(* CODESYS project FileOperation.project

Project tree, tasks and I/O mapping:
  Device : CODESYS Control for Raspberry Pi MC SL, CODESYS GmbH, order no. 2302000009, version 4.11.0.0
    application Application
      libraries: Standard, 3.5.18.0 (System); VisuDialogs, 4.5.0.0 (System); Visu Utils, 4.5.0.0 (System); CAA File, * (CAA Technical Workgroup)
      task MainTask (cyclic, interval t#20ms, priority 1, watchdog t#100ms x 1) calls TEST_FileFB, SK_FileDialogExec, Test_SK_FileDialogExec
      task VISU_TASK (cyclic, interval 100 ms, priority 31) calls VisuElems.Visu_Prg
      DialogTest/
        visualisation VS_TEST_SK_FileDialogExec
        program Test_SK_FileDialogExec [ST]
      Define/
        data type CharToStringBuffer
        data type CharCode
        data type AxisData
        data type TestCheck
        data type TestState
        data type FIX_TBL
        data type SK_FileSelectDialogVar
        data type SK_FileInfo
      FunctionBlockTest/
        program TEST_FileFB [ST]
      LIBs/
        function block SKFB_ReadFile [ST]
        function block SKFB_ReadFixTbl [ST]
        function block SKFB_WriteFile [ST]
        function block SKFB_WriteFixTbl [ST]
        program SK_FileDialogExec [ST]
        visualisation SKVS_FileSelectDialog
        function block SKFB_ListFilesInDir [ST]
    GPIOs_A_B : GPIOs A/B, 3S - Smart Software Solutions GmbH, version 4.11.0.0
        unmapped channels: digital inputs (GPIO0..GPIO31), digital outputs (GPIO0..GPIO31)
    Onewire
    Camera device
      <空>
    SPI
    I²C
    SoftMotion General Axis Pool
  text list GlobalTextList
*)

// Device/Application/Define/CharToStringBuffer
TYPE CharToStringBuffer :
UNION
	ValueBuffer: ARRAY [0..31] OF BYTE;
	ValueString: STRING;
END_UNION
END_TYPE

// Device/Application/Define/CharCode
{attribute 'qualified_only'}
{attribute 'strict'}
TYPE CharCode :
(
	NULL := 0,
	CR:= 16#0D,
	LF:= 16#0A,
	COMMA:= 16#2C	
);
END_TYPE

// Device/Application/Define/AxisData
TYPE AxisData :
STRUCT
	Value: ARRAY [0..5] OF REAL; 	//VX,VY,VZ,VA,VB,VC:REAL;
END_STRUCT
END_TYPE

// Device/Application/Define/TestCheck
TYPE TestCheck :

STRUCT
	State:TestState:= TestState.Wait;
	Msg:STRING;
END_STRUCT

END_TYPE

// Device/Application/Define/TestState
{attribute 'qualified_only'}
{attribute 'strict'}
TYPE TestState :
(
	Wait:=0, Exec:=1, Success:=10, Error:=-1
);
END_TYPE

// Device/Application/Define/FIX_TBL
TYPE FIX_TBL :
STRUCT
	Value:ARRAY[0..5,1..20] OF LREAL;
END_STRUCT
END_TYPE

// Device/Application/Define/SK_FileSelectDialogVar
TYPE SK_FileSelectDialogVar :
(*
	2024/08/02 SKVS_FileSelectDialogとやり取りする変数	
*)

STRUCT
	ListPath:STRING;//一覧で表示するパスの場所

	//FileData:ARRAY[1..SK_FileDialogExec.MAX_FILE_LISTING] OF SK_FileInfo;
	//FileCount:INT;
	Selected:INT;
	
	//Ok時に決定されたパス＋ファイル名
	//ResultPathFileName:STRING;
	////Ok時に決定されたファイル名(パスはない)
	ResultFileName:STRING;
	
	//Option_SaveMode:BOOL:=FALSE;  // 

	//Userが自由に設定できるフラグ
	//UserFlag:INT:=0;
	
	//----------------- 結果の取得 ----------------------
	
	//OKボタンで終了したらTRUE
	//DialogOK:BOOL;	
	
	//Cancelボタンで終了したらTRUE
	//DialogCancel:BOOL;
	
END_STRUCT

END_TYPE

// Device/Application/Define/SK_FileInfo
TYPE SK_FileInfo :
STRUCT
	FileName:STRING;
	FileSize:STRING;
	LastModifyDT:STRING;
END_STRUCT
END_TYPE

// Device/Application/FunctionBlockTest/TEST_FileFB
PROGRAM TEST_FileFB
(* ファイル関連のFBをテストするプログラム　*)

(* 
準備事項 RPi版 
Device-ファイルで、
ランタイム（右側）で、PlcLogicが カレントになるので、
/PlcLogic
  + /CNC_DATA
    + /LOG
    + /CONFIG
    + /GCODE

のフォルダを作製する。　
プログラムからは、　CNC_DATA/CONFIG/aaa.csv のようにアクセスする

*)

(* 
準備事項 HX版 
Device-ファイルで、
ランタイム（右側）で、SDCardが /に相当するので、
/SDCard
  + /CNC_DATA
    + /LOG
    + /CONFIG
    + /GCODE

のフォルダを作製する。
プログラムからは、　/media/sd-mmcblk0p1/CNC_DATA/CONFIG/aaa.csv のようにアクセスする
*)

VAR CONSTANT
	VAR_TBL_COUNT:INT:=20;	
	FilePath:STRING:= 'CNC_DATA/CONFIG/';	//RPi
	//FilePath:STRING:= '/media/sd-mmcblk0p1/CNC_DATA/CONFIG/';	//HITACHI HX
END_VAR	
	

VAR 	
	//GCode Table
	TBL_W:ARRAY [0..5(*AXIS*),1..VAR_TBL_COUNT] OF LREAL;
	TBL_R:ARRAY [0..5(*AXIS*),1..VAR_TBL_COUNT] OF LREAL;


	FBRead:SKFB_ReadFixTbl;
	CheckReadData:TestCheck;

	FBWriteLine:SKFB_WriteFile;
	WriteLineArray: ARRAY[0..1] OF STRING;
	CheckWriteLine:TestCheck;

	FBWrite:SKFB_WriteFixTbl;
	CheckWriteData:TestCheck;
	
	i_row,i_axis:INT;
	//Initialized:BOOL:=FALSE;
	
END_VAR


// テストシーケンス


IF (CheckWriteLine.State=TestState.Wait) THEN
	CheckWriteLine.State:= TestState.Exec;
END_IF

IF (CheckWriteLine.State=TestState.Success) AND (CheckWriteData.State= TestState.Wait) THEN
	CheckWriteData.State:=TestState.Exec;
END_IF

IF (CheckWriteData.State=TestState.Success) AND (CheckReadData.State= TestState.Wait)THEN
	CheckReadData.State:=TestState.Exec;
END_IF

(*
IF (CheckReadData.State= TestState.Wait)THEN
	CheckReadData.State:=TestState.Exec;
END_IF
*)

//--------------------   Exec Function Block   --------------------------


IF (CheckReadData.State= TestState.Exec) THEN 
	FBRead(
		pData:=ADR(TBL_R),
		DataCount:=20,
		FileName:='TEST.CSV',
		Path:=FilePath,
		xExec:=TRUE
	);
	IF(FBRead.xDone) THEN
		FBRead(xExec:=FALSE);
		CheckReadData.Msg:= FBRead.Msg;
		CheckReadData.State := TestState.Success;	
	END_IF
	IF (FBRead.xError) THEN
		FBRead(xExec:=FALSE);	
		CheckReadData.Msg:= FBRead.Msg;
		CheckReadData.State := TestState.Error;	
	END_IF
	
END_IF

IF (CheckWriteData.State= TestState.Exec) THEN
	// SetTestData
	FOR i_row:=1 TO VAR_TBL_COUNT DO
		FOR i_axis:=0 TO 5 DO
			TBL_W[i_axis,i_row]:= i_row*10+ i_axis;
		END_FOR
	END_FOR
	
	FBWrite(
		pData:=ADR(TBL_W),
		//DataCount:=20,
		FileName:='TEST.CSV',
		Path:=FilePath,
		xExec:=TRUE
	);
	IF(FBWrite.xDone) THEN
		FBWrite(xExec:=FALSE);
		CheckWriteData.Msg:= CheckWriteData.Msg;
		CheckWriteData.State := TestState.Success;	
	END_IF
	IF (FBWrite.xError) THEN
		FBWrite(xExec:=FALSE);	
		CheckWriteData.Msg:= CheckWriteData.Msg;
		CheckWriteData.State := TestState.Error;	
	END_IF
	
END_IF


IF CheckWriteLine.State= TestState.Exec THEN
	WriteLineArray[0]:='123456789$0D$0A';
	WriteLineArray[1]:='ABCDEFG$0D$0A';

	FbWriteLine(
		pWriteLines:= ADR(WriteLineArray),
		WriteLinesCount:=2,
		FilePathName:=CONCAT(FilePath,'1.TXT'),
		xExec:=TRUE
	);
	
	IF FbWriteLine.xDone THEN
		CheckWriteLine.Msg:= FbWriteLine.Msg;
		CheckWriteLine.State := TestState.Success;	
		FbWriteLine(xExec:=FALSE);
	END_IF
	IF FbWriteLine.xError THEN
		CheckWriteLine.Msg:= FbWriteLine.Msg;
		CheckWriteLine.State := TestState.Error;	
		FbWriteLine(xExec:=FALSE);
	END_IF
		
END_IF

END_PROGRAM

// Device/Application/LIBs/SKFB_ReadFixTbl
FUNCTION_BLOCK SKFB_ReadFixTbl
(*
	2024/08/02
	FixテーブルのCSVファイルを指定のバッファに読み込む
	注意:CAA File 3.5.15 を使っているため、PCエミュレーターには対応していない。　実機に転送して実行すること	
	ファイルバッファREAD_FILE_BUFFERを確保して読み込むのでファイルの大きさに注意(改善点)
*)

// Interface Variables ---------------------------------------------------

VAR_INPUT
	FileName:STRING:='';	//パスは含まない	
	Path:STRING := '';
	pData:POINTER TO FIX_TBL:=0; //データメモリへのポインタ
	DataCount:UINT:=0;  // ファイルにデータメモリ以上のデータがある場合は無視されます

	xExec:BOOL:=FALSE;	//実行・維持フラグ	
	PARSE_CHAR_COUNT:UINT:= 256;   //一度のサイクル処理でパースする文字数

END_VAR

VAR_OUTPUT
	xDone:BOOL;
	xError:BOOL;
	Msg:STRING;

	ReadRowCount: DINT; 		//読み込んだデータ数
	ExecState: INT:= stInit;	//現在の実行状況
	//DataHeader: STRING;	
END_VAR


VAR CONSTANT
	//State
	stInit:INT:=0;
	stWait:INT := 1; 
	stFileToBuffer:INT:=2;

	stParseHeader:INT:=3;
	stParseData:INT:=4;

	//Result
	stDone:INT := 100;
	stError:INT:= 999;

	//ファイルバッファ
	READ_FILE_BUFFER:UINT:=1024*16;  //バッファ	16K

END_VAR

// Implementation Variables ---------------------------------------------------


VAR
	
	FbFileRead:SKFB_ReadFile;
	RawBuff: ARRAY [0..READ_FILE_BUFFER-1] OF BYTE;	
	i_RawBuff,i_add:UINT;
	CurrBuff:BYTE;
	
	i_TempChar, i_Row, i_Axis, i_TempCharClear: INT;

	TmpCharBuffer: CharToStringBuffer;
END_VAR

CASE ExecState OF
	
	stInit:
		//初期化
		xDone:=FALSE;
		xError:=FALSE;
		Msg:='';
		FbFileRead(xExec := FALSE);
		ExecState:= stWait;
		ReadRowCount:=-1;
		
	stWait:
		IF xExec THEN
			//Exec状態になった　-->Check Input Variables 
			IF pData=0 THEN
				Msg:='pData is not set.';
				ExecState:=stError;
			ELSIF DataCount=0 THEN
				Msg:='ReadBufferSize is not set.';
				ExecState:=stError;
			ELSIF Path='' THEN
				Msg:='Path is not set.';
				ExecState:=stError;
			ELSIF FileName='' THEN
				Msg:='Path is not set.';
				ExecState:=stError;
			ELSE
				//Proceed Next State
				ExecState:= stFileToBuffer;
			END_IF
		END_IF
	
	stFileToBuffer:	// File Open
		
		FbFileRead(
			xExec:= TRUE, 
			pReadBuffer:= 		ADR(RawBuff),
			ReadBufferSize:= 	READ_FILE_BUFFER,
			FilePathName:= CONCAT(Path,FileName)
		);
	
		// Until Done or Error
		IF FbFileRead.xDone THEN
			FbFileRead(xExec := FALSE);
	
			//出力メモリのクリア
			FOR i_Row:=1 TO 20 DO
				FOR i_Axis:=0 TO 5 DO 
					pData^.Value[i_Axis,i_Row]:=0;			
				END_FOR
			END_FOR
			
			ExecState := stParseHeader;
			i_RawBuff := 0;
			i_TempChar := 0;
			i_Row := 1;
			i_Axis := 0;
			//DataHeader:='';
			
			//Clear Buffer
			FOR i_TempCharClear := 0 TO 31 DO
				TmpCharBuffer.ValueBuffer[i_TempCharClear] := 0;
			END_FOR
	
		ELSIF FbFileRead.xError THEN
			Msg:= CONCAT('FileToBuffer:',FbFileRead.Msg);
			FbFileRead(xExec := FALSE);
	
			ExecState := stError;
		END_IF

	StParseHeader:	// Skip DataTitle
		ExecState:=stParseData;

(*
	//PARSE_CHAR_COUNTづつ処理
	FOR i_add:=0 TO PARSE_CHAR_COUNT-1 DO
		IF (i_RawBuff > READ_FILE_BUFFER) THEN
			State := stError;
			Msg:= CONCAT('ParseHeader:','BUFFER OVER-RUN');	
		ELSE
			CurrBuff:=RawBuff[i_RawBuff];
			IF (CurrBuff = CharCode.LF) THEN
				DataHeader:= TmpCharBuffer.ValueString;

				//Clear Buffer
				FOR i_TempCharClear := 0 TO 31 DO
					TmpCharBuffer.ValueBuffer[i_TempCharClear] := 0;
				END_FOR
				i_TempChar:=0;
			
				State := stParseData;
				EXIT;
			ELSIF (CurrBuff = CharCode.NULL) THEN
				State := stError;
				Msg:= CONCAT('ParseHeader:','HEADER FORMAT_ERROR');	
				EXIT;
			ELSE
				//何らかの文字
				TmpCharBuffer.ValueBuffer[i_TempChar]:= CurrBuff;
				i_TempChar:=i_TempChar+1;
			END_IF;

			i_RawBuff:= i_RawBuff+1;
						
		END_IF
	END_FOR
*)
	stParseData:	
	
		//PARSE_CHAR_COUNTづつ処理
		FOR i_add:=0 TO PARSE_CHAR_COUNT-1 DO
			IF (i_RawBuff > READ_FILE_BUFFER) THEN
				ExecState := stError;
				Msg:= 'ParseData: BUFFER OVER-RUN';
			ELSE
				CurrBuff:=RawBuff[i_RawBuff];
				
				IF (CurrBuff = CharCode.COMMA) OR (CurrBuff = CharCode.CR) THEN
	
					//カンマ、もしくは改行-->値をセルに代入
					IF(i_Axis<=5) AND (i_Row<=DataCount) THEN
	
						//Buffer to Data
						pData^.Value[i_Axis,i_Row] := STRING_TO_REAL(TmpCharBuffer.ValueString);
	
						//Clear Buffer
						FOR i_TempCharClear := 0 TO 31 DO
							TmpCharBuffer.ValueBuffer[i_TempCharClear] := 0;
						END_FOR
						i_TempChar := 0;			
						
						//Next Position
						IF(CurrBuff=CharCode.COMMA) THEN
							i_Axis := i_Axis + 1;
						ELSIF (CurrBuff=CharCode.CR) THEN
							ReadRowCount:= i_Row;
							i_Row:= i_Row+1;
							i_Axis:=0;
						END_IF					
					ELSE
						IF (i_Row> DataCount) THEN
							;
							ExecState := stDone;
							Msg:= 'ParseData: Data Terminate by RowCount';					
							EXIT;
						ELSE
							//Column Over 
							ExecState := stError;
							Msg:= 'ParseData:CSV Error　: TOO MANY COLUMN';	
							EXIT;
						END_IF	
					END_IF
					
				ELSIF (CurrBuff = CharCode.LF) THEN
					//LFはCOLを0にする
					//i_Row := i_Row + 1;
					i_Axis := 0;
				ELSIF (CurrBuff = CharCode.NULL) THEN
					ExecState := stDone;
					Msg:= 'ParseData: Data Terminate by Null Char';					
					EXIT;
				ELSE
					TmpCharBuffer.ValueBuffer[i_TempChar] := RawBuff[i_RawBuff];
					i_TempChar := i_TempChar + 1;
				END_IF
				
				//Next iteration
				i_RawBuff := i_RawBuff + 1;
									
			END_IF
			
		END_FOR
	
	stDone:
		xDone:=TRUE;
		IF NOT xExec THEN
			ExecState:= stInit;
		END_IF
		
	stError:
		xError:=TRUE;
		IF NOT xExec THEN
			ExecState:= stInit;
		END_IF
		
END_CASE

END_FUNCTION_BLOCK

// Device/Application/LIBs/SKFB_ReadFile
FUNCTION_BLOCK SKFB_ReadFile
(*
	2024/08/02
	指定されたファイルを指定のバッファに読み込む
	注意:CAA File 3.5.15 を使っているため、PCエミュレーターには対応していない。　実機に転送して実行すること	
*)

// Interface Variables ---------------------------------------------------

VAR_INPUT
	pReadBuffer:POINTER TO ARRAY[0..0] OF BYTE:=0;
	ReadBufferSize:UDINT:=0;
	xExec:BOOL:=FALSE;
	FilePathName:STRING;
	ReadTimeout_InMicrosec:UDINT:= 1000;
END_VAR

VAR_OUTPUT
	xError:BOOL;
	xDone:BOOL;
	ExecState:INT := stInit;
	Msg:STRING;
END_VAR

VAR CONSTANT
	//Execute Sequence State (--> ExecState )
	stInit:INT:=0;
	stWait:INT:=1;
	stOpen:INT:=2;
	stRead:INT:=3;
	stClose:INT:=4;
	stDone:INT:=100;
	stError:INT:=999;
END_VAR

// Implementation Variables ---------------------------------------------------

VAR
	FOpenDone: BOOL;
(* HX: 
	FileHandle: CAA.HANDLE;
 *)

(* RPi: *)
	FileHandle: DWORD;
(* *)

	FB_Open: FILE.Open;
	FB_Read: FILE.Read;
	FB_Close: FILE.Close;
	FileReadSize: UDINT;
END_VAR

CASE ExecState OF
	
	stInit:
		xError:=FALSE;
		xDone:=FALSE;
		Msg:='';
		ExecState:=stWait;
	
	stWait:
		IF xExec THEN
			//Exec状態になった　-->Check Input Variables 
			IF pReadBuffer=0 THEN
				Msg:='pReadBuffer is not set.';
				ExecState:=stError;
			ELSIF ReadBufferSize=0 THEN
				Msg:='ReadBufferSize is not set.';
				ExecState:=stError;
			ELSE
				//Proceed Next State
				ExecState:=stOpen;							
			END_IF
		END_IF
	
stOpen:	// File Open
	Msg:='';
	
	FB_Open(
		xExecute:= TRUE, 
		xDone=> , 
		xBusy=> , 
		xError=> , 
		sFileName:= FilePathName,
		eFileMode:= File.MODE.MREAD, 
		xExclusive:= TRUE);

	// Until Done or Error
	IF FB_Open.xDone THEN
		FOpenDone := TRUE;
		FileHandle := FB_Open.hFile;
		FB_Open(xExecute := FALSE);
		ExecState := stRead;
	ELSIF FB_Open.xError THEN
		Msg:= CONCAT('Error:File.Open:',TO_STRING(FB_Open.eError));
		FB_Open(xExecute := FALSE);
		ExecState := stError;
	END_IF

stRead:
	FB_Read(
		xExecute:= TRUE, 
		xAbort:= , 
		udiTimeOut:= ReadTimeout_InMicrosec, //マイクロ秒=1msecでTimeout
		xDone=> , 
		xBusy=> , 
		xError=> , 
		xAborted=> , 
		hFile:= FileHandle, 
		pBuffer:= pReadBuffer, 
		szBuffer:= ReadBufferSize, 
		eError=> , 
		szSize=> FileReadSize);

	// Until Done or Error
	IF FB_Read.xDone THEN
		FB_Read(xExecute := FALSE);
		ExecState := stClose;
		Msg:= CONCAT('Success:File.Read: Size= ',TO_STRING(FileReadSize));
	ELSIF FB_Read.xError THEN
		Msg:= CONCAT('Error:File.Read:',TO_STRING(FB_Read.eError));
		FB_Read(xExecute := FALSE);
		ExecState := stError;
	END_IF

stClose:
	FB_Close(
		xExecute:= TRUE, 
		xDone=> , 
		xBusy=> , 
		xError=> , 
		hFile:= FileHandle, 
		eError=> );

	// Until Done or Error
	IF FB_Close.xDone THEN
		FB_Close(xExecute := FALSE);
		ExecState := stDone;
	ELSIF FB_Close.xError THEN
		Msg:= CONCAT('Error.File.Close:',TO_STRING(FB_Open.eError));
		FB_Close(xExecute := FALSE);
		ExecState := stError;
	END_IF

stDone:
	xDone:=TRUE;
	IF (xExec=FALSE) THEN
		ExecState:=stInit;
	END_IF

stError:
	xError:=TRUE;
	IF (xExec=FALSE) THEN
		ExecState:=stInit;
	END_IF

	
END_CASE

END_FUNCTION_BLOCK

// Device/Application/LIBs/SKFB_WriteFile
FUNCTION_BLOCK SKFB_WriteFile
(*
	2024/08/02
	指定のバッファを、指定されたファイルに書き込みます
	注意:CAA File 3.5.15 を使っているため、PCエミュレーターには対応していない。　実機に転送して実行すること	
*)

// Interface Variables ---------------------------------------------------

VAR_INPUT
	FilePathName:STRING:='';	// ファイル名（フルパス)
	xExec:BOOL:=FALSE;		// 実行・維持フラグ

	pWriteLines:POINTER TO ARRAY[0..0] OF STRING:=0;	//書き込み行バッファ(string)
	WriteLinesCount:UINT:=0;							//書き込み行バッファ数
	
	WriteTimeout_InMicrosec:UDINT:= 6000;			//書き込みタイムアウト (マイクロ秒)
	FileMode:FILE.MODE:= File.MODE.MWRITE;			//書き込み時のファイルモード
END_VAR

VAR_OUTPUT
	xError:BOOL;				// 実行結果エラー
	xDone:BOOL;					// 実行終了(OK)
	Msg:STRING;					// 実行メッセージ(エラーメッセージ)
	ExecState:INT := stInit;	// 現在実行状況
	LinesWritten:INT;			// 現在の書き込み行数
END_VAR

VAR CONSTANT
	//Execute Sequence State (--> ExecState )
	stInit:INT:=0;
	stWait:INT:=1;
	stOpen:INT:=2;
	stWrite:INT:=3;
	stClose:INT:=4;
	stDone:INT:=100;
	stError:INT:=999;
END_VAR

// Implementation Variables ---------------------------------------------------

VAR
	FOpenDone: BOOL;
(* HX: 
	FileHandle: CAA.HANDLE;
 *)

(* RPi: *)
	FileHandle: DWORD; // DWORD;
(* *)

	FB_Open: FILE.Open;
	FB_Write: FILE.Write;
	FB_Close: FILE.Close;
	i_Line:INT;
END_VAR

CASE ExecState OF
	
	stInit:
		xError:=FALSE;
		xDone:=FALSE;
		Msg:='';
		LinesWritten:=-1;
		i_Line:=0;
		ExecState:=stWait;
		
	stWait:
		IF xExec THEN
			//Exec状態になった　-->Check Input Variables 
			IF pWriteLines=0 THEN
				Msg:='pWriteLines is not set.';
				ExecState:=stError;
			ELSIF WriteLinesCount=0 THEN
				Msg:='WriteLinesCount is not set.';
				ExecState:=stError;
			ELSIF FilePathName='' THEN
				Msg:='FilePathName is not set.';
				ExecState:=stError;
			ELSE
				//Proceed Next State
				ExecState:=stOpen;							
			END_IF
		END_IF	
	
	stOpen:	// File Open
		Msg:='';
		
		FB_Open(
			xExecute:= TRUE, 
			xDone=> , 
			xBusy=> , 
			xError=> , 
			sFileName:= FilePathName,
			eFileMode:= FileMode,
			xExclusive:= TRUE);
	
		// Until Done or Error
		IF FB_Open.xDone THEN
			FOpenDone := TRUE;
			FileHandle := FB_Open.hFile;
			FB_Open(xExecute := FALSE);
			ExecState := stWrite;
		ELSIF FB_Open.xError THEN
			Msg:= CONCAT('Error:File.Open:',TO_STRING(FB_Open.eError));
			FB_Open(xExecute := FALSE);
			ExecState := stError;
		END_IF
	
	stWrite:
		FB_Write(
			xExecute:= TRUE, 
			xAbort:= , 
			udiTimeOut:= WriteTimeout_InMicrosec, //マイクロ秒=1msecでTimeout
			xDone=> , 
			xBusy=> , 
			xError=> , 
			xAborted=> , 
			hFile:= FileHandle, 
			pBuffer:= ADR(pWriteLines^[i_Line]), 
			szSize:= TO_UDINT( LEN(pWriteLines^[i_Line]) )
		);
	
		// Until Done or Error
		IF FB_Write.xDone THEN
			LinesWritten:= i_Line+1;
			
			IF(i_Line>=WriteLinesCount-1) THEN			
				Msg:= CONCAT('Finish WriteFile : WrittenLineCount= ',TO_STRING(LinesWritten));
				ExecState := stClose;
			ELSE
				Msg:= CONCAT('WriteFile LineCount= ',TO_STRING(LinesWritten));
				i_Line:= i_Line+1;
			END_IF
	
			FB_Write(xExecute := FALSE);
	
		ELSIF FB_Write.xError THEN
			Msg:= CONCAT('Error:File.Write:',TO_STRING(FB_Write.eError));
			FB_Write(xExecute := FALSE);
			ExecState := stError;
		END_IF
	
	stClose:
		FB_Close(
			xExecute:= TRUE, 
			xDone=> , 
			xBusy=> , 
			xError=> , 
			hFile:= FileHandle, 
			eError=> );
	
		// Until Done or Error
		IF FB_Close.xDone THEN
			FB_Close(xExecute := FALSE);
			ExecState := stDone;
		ELSIF FB_Close.xError THEN
			Msg:= CONCAT('Error.File.Close:',TO_STRING(FB_Open.eError));
			FB_Close(xExecute := FALSE);
			ExecState := stError;
		END_IF
	
	stDone:
		xDone:=TRUE;
		IF (xExec=FALSE) THEN
			ExecState:=stInit;
		END_IF
	
	stError:
		xError:=TRUE;
		IF (xExec=FALSE) THEN
			ExecState:=stInit;
		END_IF
	
	
END_CASE

END_FUNCTION_BLOCK

// Device/Application/LIBs/SKFB_WriteFixTbl
FUNCTION_BLOCK SKFB_WriteFixTbl
(*
	2024/08/02
	Fixテーブルを、指定のファイルにCSVとして書き込む
	注意:CAA File 3.5.15 を使っているため、PCエミュレーターには対応していない。　実機に転送して実行すること	
*)

// Interface Variables ---------------------------------------------------

VAR_INPUT
	FileName:STRING:='';   //パスは含まない形のファイル名	
	Path:STRING := '';     //パス　フォルダの最後のスラッシュが必要
	xExec:BOOL:=FALSE;				//実行/維持フラグ	
	pData:POINTER TO FIX_TBL:=0; 	//FIX_TBL構造体へのポインタ
END_VAR

VAR_OUTPUT
	Msg:STRING;
	xDone:BOOL;
	xError:BOOL;
END_VAR

VAR CONSTANT
	//Execute Sequence State (--> ExecState )
	stInit:INT:=0;
	stWait:INT := 1; 
	stDataToBuffer:INT :=2;
	stWriteFile:INT:=3;

	//Result
	stDone:INT := 100;
	stError:INT:= 999;

	//ファイルバッファ
	MAX_WRITE_LINE:UINT:=20;  //バッファ	20行	(FIX_TBLの行数)
END_VAR

// Implementation Variables ---------------------------------------------------



VAR
	State: INT:= stInit;	
	FbFileWrite:SKFB_WriteFile;
	Lines:ARRAY[0..MAX_WRITE_LINE-1] OF STRING; //  FIX_TBLの行数を確保
	i_RawBuff:UINT;
	i_Row: INT;
	i_Axis:INT;
	str_ax:STRING;
	str_line:STRING;
END_VAR

CASE State OF
	
	stInit:
		xDone:=FALSE;
		xError:=FALSE;
		Msg:='';
		FbFileWrite(xExec := FALSE);
		State:= stWait;
		i_Row:=1;
		i_RawBuff:=0;
		
	stWait:
		IF xExec THEN
			IF pData=0 THEN
				Msg:='pData is not set.';
				State:=stError;
			ELSIF (CONCAT(Path,FileName)='') THEN
				Msg:='Path and Filename are not set.';
				State:=stError;
			ELSE
				State:= StDataToBuffer;					
			END_IF
			
		END_IF
		
	stDataToBuffer:
		// 1行づつ処理
		str_line:='';
		FOR i_Axis:=0 TO 5 DO
			str_ax:= TO_STRING(pData^.Value[i_Axis,i_Row]);	
			str_line:= CONCAT(str_line, str_ax);
			IF i_Axis<5 THEN
				str_line:=CONCAT(str_line,',');
			ELSE
				str_line:=CONCAT(str_line,'$0D$0A');
			END_IF	
		END_FOR
		//str_lineを加える
		Lines[i_Row-1]:= str_line;
		
		
		//for Next Row
		IF i_Row = MAX_WRITE_LINE THEN
			State:= StWriteFile;
		ELSE
			i_Row:=i_Row+1;	
		END_IF
		
		
	stWriteFile:	// File Write
		
		FbFileWrite(
			xExec:= TRUE, 
			pWriteLines:= ADR(Lines),
			WriteLinesCount:= MAX_WRITE_LINE,
			FilePathName:= CONCAT(Path,FileName),
		);
	
		// Until Done or Error
		IF FbFileWrite.xDone THEN
			FbFileWrite(xExec := FALSE);
	
			State := StDone;
		ELSIF FbFileWrite.xError THEN
			Msg:= CONCAT('Error FileToBuffer:',FbFileWrite.Msg);
			FbFileWrite(xExec := FALSE);
	
			State := stError;
		END_IF
	
	stDone:
		xDone:=TRUE;
		IF NOT xExec THEN
			State:= stInit;
		END_IF
		
	stError:
		xError:=TRUE;
		IF NOT xExec THEN
			State:= stInit;
		END_IF
	
END_CASE

END_FUNCTION_BLOCK

// Device/Application/LIBs/SK_FileDialogExec
PROGRAM SK_FileDialogExec
(*
	2024/08/08-2
	SKVS_FileSelectDialogの実行タスク、画面とセットで使う
*)

// Interface Variables ---------------------------------------------------
VAR CONSTANT
	MAX_FILE_LISTING:UINT:=30;
END_VAR

VAR_INPUT
	//ダイアログを実行する( メイン側のボタンに記述 )
	xExec:BOOL;	
	ListPath:STRING:='';		//	リストするパス
	UserFlag:INT:=0; 		//	呼び出した側の記録用(　呼び出しが複数ある場合、何のために呼び出したか？）
	SaveMode:BOOL:=FALSE;	//  Trueにすると、既存ファイルを選択するだけではなく、自分で新しくファイル名を入力することができる
	DefaultFileName:STRING; //	デフォルトの名前を設定したい場合に使用(SaveMode=TRUEの時)
END_VAR

VAR_OUTPUT
	
	xError:BOOL;
	xDone:BOOL;

	//Result_はxDone=TRUEの時に有効な出力
	Result_Ok:BOOL;		
	Result_Cancel:BOOL; 

	//現在の実行状態
	ExecState:INT:=0;
	//エラーなど
	Msg:STRING;

	//Okを押された時のパスファイル名 Cancelの時は"" (ただし、Okの時も""となる=何も選択していない可能性もある)
	Result_PathFileName:STRING;
	Result_FileName:STRING; // ファイル名のみ
	
END_VAR

VAR CONSTANT
	//Execute Sequence State (--> ExecState )
	stInit:INT:=0;
	stWait:INT:=1;
	stListFile:INT:=2;
	stSetDialogVar:INT:=3;
	stOpenDialog:INT:=4;
	stProcessDialog:INT:=5;
	
	stResultOK:INT:=100;
	stResultCancel:INT:=200;

	stDone:INT:=300;
	stError:INT:=999;
END_VAR

// Implementation Variables ---------------------------------------------------

VAR
	PrevExecDialog:BOOL:=FALSE;	//立ち上がり検出用

	FBListFile:SKFB_ListFilesInDir;		//Dir内のファイルをリストする
	ListedFiles:ARRAY[0..MAX_FILE_LISTING-1] OF File.FILE_DIR_ENTRY; //リストされたデータ
	ListedCount:INT;
	
	Dialog_FileData:ARRAY[1..MAX_FILE_LISTING] OF SK_FileInfo;
	Dialog_FileCount:INT;
	Dialog_SelectedIndex:INT;
	Dialog_FileName:STRING;

	// ダイアログと交換するデータ
	i_listed:INT;
	i_FileData:INT;
	PrevSelected:INT:=-100;
	//Open_FileDialog:BOOL; 					//ファイル選択ダイアログ実行中
	FBOpenDialog : VU.FbOpenDialogExtended;			//ダイアログを開くFB
	DialogVars : SKVS_FileSelectDialog_VISU_STRUCT;	//Var引数とやりとりする変数 (VS名+"_VISU_STRUCT"　で自動定義される)
	WaitClosed:BOOL;	// TRUE = OkかCancelを待っている状態
	
	DialogResult_OK:BOOL;
	DialogResult_Cancel:BOOL;
END_VAR

//立ち下がり信号で処理中の場合もリセット
IF NOT xExec AND PrevExecDialog THEN

	IF(ExecState<stDone) THEN
		ExecState:=stInit;
		Msg:='xExec=>false while processing. Init Process State.';
	END_IF

END_IF;
PrevExecDialog:= xExec;


CASE ExecState OF
	stInit:
		// Clear/Init Output
		Result_Ok:=FALSE;
		Result_Cancel:=FALSE;
		xError:=FALSE;
		xDone:=FALSE;
		Result_PathFileName:='';  // Clear.
		Result_FileName:='';
		ExecState:=1;
		Msg:='';
		
	stWait:
		IF( xExec ) THEN
			//立ち上がり
			IF(ListPath='') THEN
				Msg:='ListPath is not set.';
				ExecState:=stError;
			ELSE
				ExecState:=stListFile;					
			END_IF						
		END_IF
		
	stListFile:

		//ファイルの列挙FB-- SKFB_ListFilesInDir（継続)
		FBListFile(
			ListPath:= ListPath,
			pFileInfoArray:= ADR(ListedFiles),
			FileInfoCount:= TO_INT(MAX_FILE_LISTING), //MAX=30
			xExec:=TRUE
		);	
		
		//ファイルの列挙終了判定
		IF(FBListFile.xDone)THEN
			FBListFile(xExec:=FALSE);
			i_FileData:=0;
			FOR i_listed:=0 TO FBListFile.ListedCount-1 DO 
				IF ListedFiles[i_listed].xDirectory=FALSE THEN
					i_FileData:=i_FileData+1;	//先にIncして、Indexを1..30に。 = ファイルの1列目の番号を1からはじめたい。	
					Dialog_FileData[i_FileData].FileName:= 	ListedFiles[i_listed].sEntry;
					Dialog_FileData[i_FileData].FileSize:= 	TO_STRING(ListedFiles[i_listed].szSize);
					Dialog_FileData[i_FileData].LastModifyDT:= TO_STRING(ListedFiles[i_listed].dtLastModification);	
				END_IF
			END_FOR
			
			ListedCount:= i_FileData;
			Dialog_FileCount:= i_FileData;
			Dialog_FileName:=DefaultFileName;
			Dialog_SelectedIndex:=0;		//No Selection.

			// Next.
			ExecState:=stSetDialogVar;
		END_IF
		
		IF(FBListFile.xError)THEN
			FBListFile(xExec:=FALSE);
			Msg:= CONCAT('Check FileDirectory of Device = ',ListPath);
			ExecState:=stError;
		END_IF
		
	stSetDialogVar:
		//Set DialogVars
		DialogVars.FileArrayPtr		:=ADR(Dialog_FileData);
		DialogVars.FileArrayCount	:=Dialog_FileCount;
		DialogVars.ListPath			:=ListPath;
		
		IF SaveMode=TRUE THEN
			DialogVars.Mode				:=1;  // SaveMode
		ELSE
			DialogVars.Mode				:=0;  // SelectMode
		END_IF
	
		DialogResult_OK:=FALSE;
		DialogResult_Cancel:=FALSE;	
		
		DialogVars.DialogOK REF= DialogResult_OK;//DialogData.DialogOK;
		DialogVars.DialogCancel REF= DialogResult_Cancel;//DialogData.DialogCancel;
		DialogVars.FileSelectedIndex REF= Dialog_SelectedIndex;
		DialogVars.SaveFileName REF= Dialog_FileName;  // 初期のファイル名
		WaitClosed:=TRUE;
		ExecState:=stOpenDialog;
		
	stOpenDialog:
		//OpenModal (起動中)
		FBOpenDialog(
			sDialogName := 'SKVS_FileSelectDialog', //開きたいダイアログの名前
			xModal := TRUE, 
			pTopLeftPosition := 0, 
			itfClientFilter := VU.Globals.AllClients,
			xExecute := TRUE, 
			pbyDialogInterfaceData := ADR(DialogVars), 
			udiDialogInterfaceDataSize := SIZEOF(DialogVars));
			
		IF FBOpenDialog.xDone OR FBOpenDialog.xError THEN
			//Next Jump
			IF (FBOpenDialog.xDone) THEN
				ExecState:=stProcessDialog;
			ELSE
				ExecState:=stError;
			END_IF
			FBOpenDialog(xExecute:=FALSE);			
		END_IF

	stProcessDialog:	//ダイアログの実行中( Cancel or Okが押されるまで継続 )
		IF DialogVars.FileSelectedIndex<> PrevSelected THEN
			// ダイアログの選択が変化したら、ファイル名を設定する。 SaveDialog時には選択したファイル名を元に、新しいファイル名を作るなどできる。	
			IF(DialogVars.FileSelectedIndex)>0 THEN
				DialogVars.SaveFileName:=Dialog_FileData[DialogVars.FileSelectedIndex].FileName;
			ELSE		
				DialogVars.SaveFileName:='';
			END_IF
			PrevSelected:=DialogVars.FileSelectedIndex;
		END_IF
		
		(* これをするとおかしくなる
		IF(DialogVars.FileSelectedIndex)>0 THEN
			//選択と一致しないかどうか（文字入力・変更があった場合）
			IF DialogVars.SaveFileName<>DialogData.FileData[DialogVars.FileSelectedIndex].FileName THEN
				DialogVars.FileSelectedIndex:=0;
			END_IF		
		END_IF
		*)

		IF DialogResult_OK THEN
			ExecState:=stResultOK;
		END_IF
			
		IF DialogResult_Cancel THEN
			ExecState:=stResultCancel;
		END_IF

	stResultOK:  
		// OK Pressed. --> SetResult
		IF DialogVars.SaveFileName<>'' THEN
			Result_FileName:=DialogVars.SaveFileName;
			Result_PathFileName:= 
				CONCAT(ListPath,Result_FileName);
		END_IF
		Result_Ok:=TRUE;
		ExecState:=stDone;

	stResultCancel:
		Result_Cancel:=TRUE;
		ExecState:=stDone;
		
	stDone:
		xDone:=TRUE;
		IF xExec=FALSE THEN
			ExecState:=stInit;
		END_IF

	stError: //Error
		xError:=TRUE;	
		IF xExec=FALSE THEN
			ExecState:=stInit;
		END_IF
END_CASE

END_PROGRAM

// Device/Application/LIBs/SKFB_ListFilesInDir
FUNCTION_BLOCK SKFB_ListFilesInDir
(*
	2024/08/02
	指定フォルダのファイル名などの情報を列挙して、指定のバッファに格納するFB	
	注意:CAA File 3.5.15 を使っているため、PCエミュレーターには対応していない。　実機に転送して実行すること	
*)


// Interface Variables ---------------------------------------------------

VAR_INPUT
	ListPath:STRING;	//リストするPath
	xExec:BOOL;  		//実行維持フラグ

	pFileInfoArray:POINTER TO ARRAY [0..0] OF  FILE.FILE_DIR_ENTRY:=0; // ListPathのファイル情報を受け取るバッファ
	FileInfoCount:INT:=0; // ファイル情報バッファの確保数	
END_VAR


VAR_OUTPUT
	xDone:BOOL;		//正常終了フラグ
	xError:BOOL;	//異常終了フラグ
	ExecState: INT:=stInit; //現在の実行状況
	Msg:STRING;		//
	ListedCount:INT;	//リストしたデータの数
END_VAR

VAR CONSTANT
	//Execute Sequence State (--> ExecState )
	stInit:INT:=0;
	stWait:INT:=1;
	stOpen:INT:=2;
	stList:INT:=3;
	stClose:INT:=4;
	stDone:INT:=10;
	stError:INT:=99;
END_VAR


// Implementation Variables ---------------------------------------------------

VAR
(* HX: 
	hDir: CAA.HANDLE;
 *)

(* RPi: *)
	hDir: DWORD;
(* *)
	
	dirOpen: FILE.DirOpen;
	dirList: FILE.DirList;
	dirClose: FILE.DirClose;

	i_FileInfo: INT;
	FileData1: FILE.FILE_DIR_ENTRY;
	
END_VAR


CASE ExecState OF

	stInit:
		xError:=FALSE;
		xDone:=FALSE;
		Msg:='';
		ExecState:=stWait;

	stWait:
		IF(xExec)THEN
			//Exec状態になった　-->Check Input Variables 
			IF pFileInfoArray=0 THEN
				Msg:='pFileInfoArray is not set.';
				ExecState:=stError;
			ELSIF FileInfoCount=0 THEN
				Msg:='FileInfoCount is not set.';
				ExecState:=stError;
			ELSE
				//Proceed Next State
				ExecState:=stOpen;							
			END_IF
		END_IF

	stOpen:		
		//init Counter
		i_FileInfo:=0;
		ListedCount:=0;
		//ディレクトリをオープンして、列挙
		dirOpen(
			xExecute:= TRUE, 
			xDone=> , 
			xBusy=> , 
			xError=> , 
			sDirName:= ListPath,
	
			eError=> , 
			hDir=> );
		IF dirOpen.xDone THEN
			hDir := dirOpen.hDir;
			dirOpen(xExecute:= FALSE);
			ExecState := stList;
		ELSIF dirOpen.xError THEN
			Msg:=CONCAT('Error in dirOpen, ListPath=',ListPath);
			ExecState:=stError;
		END_IF
		
	stList:
	
		//エラー（NO_MORE_ENTRIES)になるまで何度か繰り返す必要がある
		dirList(
			xExecute:= TRUE, 
			xDone=> , 
			xBusy=> , 
			xError=> , 
			hDir:= hDir, 
			eError=> , 
			deDirEntry=> FileData1);
			
		//ERRORチェック
		IF dirList.xError THEN
			IF (dirList.eError = FILE.ERROR.NO_MORE_ENTRIES) THEN
				//リストし終えたので終了
				Msg:='Success all LISTED.';
				ExecState := stClose; 		
			ELSE
				//その他通常のエラー
				Msg:=CONCAT('ERROR in dirList: ',TO_STRING(dirList.eError));
				ExecState:=stError;
			END_IF
			dirList(xExecute:= FALSE);		//これをするとeErrorが NO_ERRORになる			
		END_IF

		//取得した１データを格納
		IF dirList.xDone THEN
			dirList(xExecute:= FALSE);
			IF i_FileInfo<FileInfoCount THEN
				pFileInfoArray^[i_FileInfo] := FileData1;
				i_FileInfo := i_FileInfo + 1;
				ListedCount:=i_FileInfo;			
			ELSE
				//最大数をオーバーしたので終了
				Msg:='Listing OVER FileInfoCount';
				ExecState:=stClose;
			END_IF
		END_IF
		
	stClose:
		dirClose(
			xExecute:= TRUE, 
			xDone=> , 
			xBusy=> , 
			xError=> , 
			hDir:= hDir, 
			eError=> );

		IF dirClose.xDone THEN
			dirClose(xExecute:= FALSE);
			hDir := 0;
			ExecState := stDone; 
		END_IF

		IF dirClose.xError THEN
			Msg:=CONCAT('ERROR:DirClose:',TO_STRING(dirClose.eError));
			dirClose(xExecute:= FALSE);
			hDir := 0;
			ExecState := stError; 
		END_IF
		
	stDone:
		//Ok
		xDone:=TRUE;
		IF(xExec=FALSE)THEN
			ExecState:= stInit;
		END_IF
	
	stError:
		//Error発生
		xError:=TRUE;
		IF(xExec=FALSE)THEN
			ExecState:= stInit;
		END_IF
					
END_CASE

END_FUNCTION_BLOCK

// Device/Application/DialogTest/Test_SK_FileDialogExec
PROGRAM Test_SK_FileDialogExec //ファイルダイアログをCNC用に使えるようにします
VAR
	Initialized:BOOL:=FALSE;
	ManualMode:BOOL:=TRUE;
	AutoResult:STRING;
END_VAR

IF NOT Initialized THEN
	SK_FileDialogExec.ListPath:=Test_FileFB.FilePath;
	Initialized:=TRUE;	
END_IF

IF ManualMode THEN
	RETURN;
END_IF

//ダイアログデータがOkの時 

IF Sk_FileDialogExec.xExec AND Sk_FileDialogExec.xDone THEN
	IF Sk_FileDialogExec.Result_Cancel THEN
		//TODO CANCELのログ
		;
		AutoResult:= CONCAT( INT_TO_STRING(SK_FileDialogExec.UserFlag),' / Canceled.'); 		
	ELSE
		AutoResult:= CONCAT( CONCAT( INT_TO_STRING(SK_FileDialogExec.UserFlag),' / Ok. FileName ='),Sk_FileDialogExec.Result_FileName); 		

		//キャンセルじゃなければ読み込み処理など
		(*
		IF Sk_FileDialogExec.UserFlag= TCNCFileDialogType.GCodeRead THEN 

			//Gコードを設定(パス＋ファイル)
			CNC.PgmFileName:=Sk_FileDialogExec.Result_PathFileName;
			CNC.PgmFileChanged:=TRUE;
		
		ELSE
	
			//補正ファイル名(ファイル名のみ)
			CNC_FixTable_Func.FileName:= Sk_FileDialogExec.Result_FileName;
	
			//コマンドを設定			
			CASE Sk_FileDialogExec.UserFlag OF
				TCNCFileDialogType.FixG54Read:
					CNC_FixTable_Func.Cmd:= CNC_FixTable_Func.CMD_G54_LOAD;
				TCNCFileDialogType.FixG54Write:
					CNC_FixTable_Func.Cmd:= CNC_FixTable_Func.CMD_G54_SAVE;
				TCNCFileDialogType.FixToolRead:
					CNC_FixTable_Func.Cmd:= CNC_FixTable_Func.CMD_TOOL_LOAD;
				TCNCFileDialogType.FixToolWrite:
					CNC_FixTable_Func.Cmd:= CNC_FixTable_Func.CMD_TOOL_SAVE;			
			END_CASE
		END_IF
		*)	
	END_IF
	
	//ファイルダイアログの実行終了
	Sk_FileDialogExec.xExec:=FALSE;
END_IF

END_PROGRAM

// Device/Application/LIBs/SKVS_FileSelectDialog
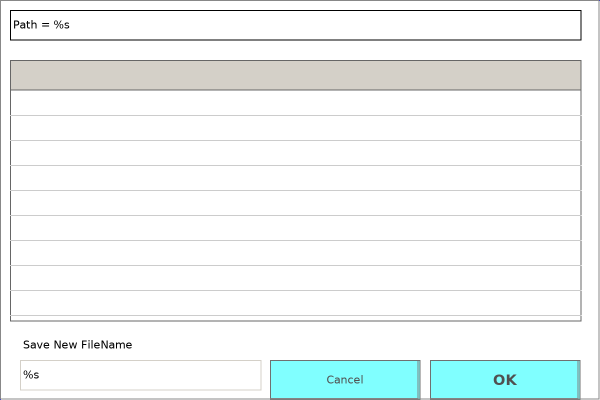
VISUALIZATION SKVS_FileSelectDialog  // 600x400
VAR_INPUT
	FileArrayPtr:POINTER TO ARRAY[1..30] OF SK_FileInfo;
	FileArrayCount:INT;
	ListPath:STRING;	
	Mode:INT :=0;  // 0= Load 1=Save
END_VAR

VAR_IN_OUT
	{attribute 'VAR_IN_OUT_AS_POINTER'}
	FileSelectedIndex:INT;
	{attribute 'VAR_IN_OUT_AS_POINTER'}
	DialogOK:BOOL;
	{attribute 'VAR_IN_OUT_AS_POINTER'}
	DialogCancel:BOOL;
	{attribute 'VAR_IN_OUT_AS_POINTER'}
	SaveFileName:STRING;
END_VAR
    Rectangle (0,0 601x421)
    Rectangle (10,10 571x30), "Path = %s", text variable: ListPath
    Button (270,360 150x40), "Cancel"
        OnMouseClick: execute { FileSelectedIndex:=-1; DialogCancel:=TRUE; }
        OnMouseClick:  Dialog=SKVS_FileSelectDialog, Result=Cancel, NumpadKeypadSet=True
    Button (430,360 150x40), "OK"
        OnMouseClick: execute { DialogOK:=TRUE; }
        OnMouseClick:  Dialog=SKVS_FileSelectDialog, Result=OK, NumpadKeypadSet=True
    Table (10,60 571x261), data array: FileArrayPtr^
        p2170511999: HX_FileSelect.str[INDEX].xExclusive
        p3723444502: HX_FileSelect.str[INDEX].dtLastModification
        p1218418051: HX_FileSelect.FileNames[5,INDEX]
        p746581629: HX_FileSelect.FileNames[6,INDEX]
        p3104783080: HX_FileSelect.FileNames[7,INDEX]
        p2501879983: HX_FileSelect.FileNames[8,INDEX]
        p7306298: HX_FileSelect.FileNames[9,INDEX]
        p1933151965: HX_FileSelect.FileNames[10,INDEX]
        p3863566920: HX_FileSelect.FileNames[11,INDEX]
        p2192122294: HX_FileSelect.FileNames[12,INDEX]
        p400160035: HX_FileSelect.FileNames[13,INDEX]
        p1265227338: HX_FileSelect.FileNames[14,INDEX]
        p3726181087: HX_FileSelect.FileNames[15,INDEX]
        p3136911649: HX_FileSelect.FileNames[16,INDEX]
        p797552052: HX_FileSelect.FileNames[17,INDEX]
        p60375027: HX_FileSelect.FileNames[18,INDEX]
        p2531912550: HX_FileSelect.FileNames[19,INDEX]
        p693678525: HX_FileSelect.FileNames[20,INDEX]
        p3156763944: HX_FileSelect.FileNames[21,INDEX]
        p3636993750: HX_FileSelect.FileNames[22,INDEX]
        p1303956035: HX_FileSelect.FileNames[23,INDEX]
        p285796650: HX_FileSelect.FileNames[24,INDEX]
        p2222472639: HX_FileSelect.FileNames[25,INDEX]
        p3768075841: HX_FileSelect.FileNames[26,INDEX]
        p1978176212: HX_FileSelect.FileNames[27,INDEX]
        p1509425299: HX_FileSelect.FileNames[28,INDEX]
        p3431519238: HX_FileSelect.FileNames[29,INDEX]
        p2846402210: HX_FileSelect.FileNames[30,INDEX]
        p1020817975: HX_FileSelect.FileNames[31,INDEX]
        p1480067529: HX_FileSelect.FileNames[32,INDEX]
        p3444104540: HX_FileSelect.FileNames[33,INDEX]
        p2449014325: HX_FileSelect.FileNames[34,INDEX]
        p76032672: HX_FileSelect.FileNames[35,INDEX]
        p1617449310: HX_FileSelect.FileNames[36,INDEX]
        p4112025035: HX_FileSelect.FileNames[37,INDEX]
        p3641186188: HX_FileSelect.FileNames[38,INDEX]
        p1282982681: HX_FileSelect.FileNames[39,INDEX]
        p2644168573: HX_FileSelect.FileNames[40,INDEX]
        p149560296: HX_FileSelect.FileNames[41,INDEX]
        p1812619286: HX_FileSelect.FileNames[42,INDEX]
        p4185568387: HX_FileSelect.FileNames[43,INDEX]
        p2781517802: HX_FileSelect.FileNames[44,INDEX]
        p817513343: HX_FileSelect.FileNames[45,INDEX]
        p1415198849: HX_FileSelect.FileNames[46,INDEX]
        p3240815636: HX_FileSelect.FileNames[47,INDEX]
        p3980033619: HX_FileSelect.FileNames[48,INDEX]
        p2018159302: HX_FileSelect.FileNames[49,INDEX]
        p493541474: HX_FileSelect.FileNames[50,INDEX]
        p2283408631: HX_FileSelect.FileNames[51,INDEX]
        p3975837449: HX_FileSelect.FileNames[52,INDEX]
        p2039128988: HX_FileSelect.FileNames[53,INDEX]
        p624591093: HX_FileSelect.FileNames[54,INDEX]
        p2957661280: HX_FileSelect.FileNames[55,INDEX]
        p3567923102: HX_FileSelect.FileNames[56,INDEX]
        p1104870155: HX_FileSelect.FileNames[57,INDEX]
        p1841981772: HX_FileSelect.FileNames[58,INDEX]
        p4172987865: HX_FileSelect.FileNames[59,INDEX]
        p1191962370: HX_FileSelect.FileNames[60,INDEX]
        p3531289495: HX_FileSelect.FileNames[61,INDEX]
        p3063629929: HX_FileSelect.FileNames[62,INDEX]
        p602643708: HX_FileSelect.FileNames[63,INDEX]
        p2136719253: HX_FileSelect.FileNames[64,INDEX]
        p3928713984: HX_FileSelect.FileNames[65,INDEX]
        p2395672830: HX_FileSelect.FileNames[66,INDEX]
        p465290347: HX_FileSelect.FileNames[67,INDEX]
        p933975596: HX_FileSelect.FileNames[68,INDEX]
        p2732294841: HX_FileSelect.FileNames[69,INDEX]
        p3355176989: HX_FileSelect.FileNames[70,INDEX]
        p1384850568: HX_FileSelect.FileNames[71,INDEX]
        p913006454: HX_FileSelect.FileNames[72,INDEX]
        p2736491491: HX_FileSelect.FileNames[73,INDEX]
        p4289439882: HX_FileSelect.FileNames[74,INDEX]
        p1792769055: HX_FileSelect.FileNames[75,INDEX]
        p238749665: HX_FileSelect.FileNames[76,INDEX]
        p2605437812: HX_FileSelect.FileNames[77,INDEX]
        p3076210995: HX_FileSelect.FileNames[78,INDEX]
        p573281702: HX_FileSelect.FileNames[79,INDEX]
        p795817148: HX_FileSelect.FileNames[80,INDEX]
        p3122651177: HX_FileSelect.FileNames[81,INDEX]
        p3741293527: HX_FileSelect.FileNames[82,INDEX]
        p1267683138: HX_FileSelect.FileNames[83,INDEX]
        p390032427: HX_FileSelect.FileNames[84,INDEX]
        p2186262718: HX_FileSelect.FileNames[85,INDEX]
        p3870278464: HX_FileSelect.FileNames[86,INDEX]
        p1944000469: HX_FileSelect.FileNames[87,INDEX]
        p1607435666: HX_FileSelect.FileNames[88,INDEX]
        p3401535751: HX_FileSelect.FileNames[89,INDEX]
        p2946442147: HX_FileSelect.FileNames[90,INDEX]
        p988804918: HX_FileSelect.FileNames[91,INDEX]
        p1578077384: HX_FileSelect.FileNames[92,INDEX]
        p3414120541: HX_FileSelect.FileNames[93,INDEX]
        p2546957108: HX_FileSelect.FileNames[94,INDEX]
        p46116769: HX_FileSelect.FileNames[95,INDEX]
        p1717556319: HX_FileSelect.FileNames[96,INDEX]
        p4079943882: HX_FileSelect.FileNames[97,INDEX]
        p3745485453: HX_FileSelect.FileNames[98,INDEX]
        p1246709272: HX_FileSelect.FileNames[99,INDEX]
        p1014161805: 30 - 1 + 1
        p1128707560: FileArrayCount
        p1137915858: FileSelectedIndex
        p3854506369: FileArrayPtr^[INDEX].FileName
        p1892666644: FileArrayPtr^[INDEX].FileSize
        p338671338: FileArrayPtr^[INDEX].LastModifyDT
        p1755163831: LastModifiedDT
    Label (20,330 150x30), "Save New FileName", invisible if: Mode=0
    Textfield (20,360 241x30), "%s", text variable: SaveFileName, invisible if: Mode=0
        OnMouseClick: write the text variable via Edit
END_VISUALIZATION

// Device/Application/DialogTest/VS_TEST_SK_FileDialogExec
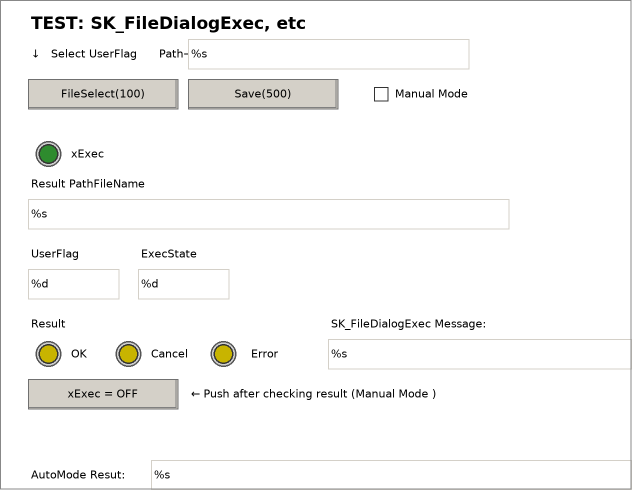
VISUALIZATION VS_TEST_SK_FileDialogExec  // 632x490
    Button (28,79 150x30), "FileSelect(100)"
        OnMouseClick: execute {
            SK_FileDialogExec.UserFlag:=100;
            SK_FileDialogExec.SaveMode:=FALSE;
            SK_FileDialogExec.xExec:=TRUE;
        }
    Textfield (28,199 481x30), "%s", text variable: SK_FileDialogExec.Result_PathFileName
    Button (188,79 150x30), "Save(500)"
        OnMouseClick: execute {
            SK_FileDialogExec.UserFlag:=500;
            SK_FileDialogExec.SaveMode:=TRUE;
            SK_FileDialogExec.xExec:=TRUE;
        }
    Textfield (28,269 91x30), "%d", text variable: SK_FileDialogExec.UserFlag
    Label (28,169 150x30), "Result PathFileName"
    Label (28,239 81x30), "UserFlag"
    Lamp1 (28,339 41x30), variable: SK_FileDialogExec.Result_Ok, style: Lamp-Lamp1-Yellow
    Lamp1 (108,339 41x30), variable: SK_FileDialogExec.Result_Cancel, style: Lamp-Lamp1-Yellow
    Lamp1 (208,339 31x30), variable: SK_FileDialogExec.xError, style: Lamp-Lamp1-Yellow
    Textfield (138,269 91x30), "%d", text variable: SK_FileDialogExec.ExecState
    Label (138,239 91x30), "ExecState"
    Label (68,339 61x30), "OK"
    Label (148,339 61x30), "Cancel"
    Label (248,339 61x30), "Error"
    Button (28,379 150x30), "xExec = OFF"
        OnMouseClick: execute { SK_FileDialogExec.xExec:=FALSE; }
    Lamp1 (28,139 41x30), variable: SK_FileDialogExec.xExec, style: Lamp-Lamp1-Green
    Label (68,139 61x30), "xExec"
    Label (188,379 261x30), "← Push after checking result (Manual Mode )"
    Label (28,309 91x30), "Result"
    Label (28,39 219x30), "↓ Select UserFlag Path→"
    Textfield (328,339 304x30), "%s", text variable: SK_FileDialogExec.Msg
    Checkbox (372,79 150x30), "Manual Mode", variable: Test_SK_FileDialogExec.ManualMode
    Textfield (151,460 481x30), "%s", text variable: Test_SK_FileDialogExec.AutoResult
    Label (28,460 101x30), "AutoMode Resut:"
    Label (328,309 162x30), "SK_FileDialogExec Message:"
    Textfield (188,39 281x30), "%s", text variable: SK_FileDialogExec.ListPath
    Label (28,8 318x30), "TEST: SK_FileDialogExec, etc"
END_VISUALIZATION
